//	This Function Block Performs A Linear Interpolation 
//	It Uses Multiple Data Points On Which A Line Graph Can Be Plotted
//	Between Each Two Data Points, A Line Equation Exists
//	The Linear Interpolation Formula Can Then Be Used To Find A Sensor Output Value 

FUNCTION_BLOCK Sensor_Calibration_Multipoint
VAR_INPUT
	Sensor_Input_Value		:		REAL	:=	0.0;
	
	Start_Calibration		:		BOOL	:=	FALSE;
	Reset_Calibration		:		BOOL	:=	FALSE;
END_VAR
VAR_OUTPUT
	Calibrated_Output_Value	:		REAL	:=	0.0;
END_VAR
VAR	
	// Lookup Table
	Sensor_Points			:		ARRAY[1..Calibration_Points] OF REAL	:=	[0.00, 25.00, 50.00, 75.00, 100.0];		//	Sensor Input - Will Be supplied From Analogue Scaling Block
	Reference_Points		:		ARRAY[1..Calibration_Points] OF REAL	:=	[0.00, 30.55, 58.16, 69.09, 100.0];		//	Actual Value
	
	Calibration_Index		: 		UINT;
	
	//	Linear Line Equation Variables
	X1						:		REAL	:=	0.0;
	X2						:		REAL	:=	0.0;
	Y1						:		REAL	:=	0.0;
	Y2						:		REAL	:=	0.0;	
END_VAR
VAR CONSTANT
	Calibration_Points		:		UINT	:=	5;
END_VAR

IF(Start_Calibration)THEN
	FOR Calibration_Index := 1 TO Calibration_Points DO
		//	Determine Between Which Two Data Points The Sensors Value Lies
		IF(Sensor_Input_Value >= Sensor_Points[Calibration_Index] AND Sensor_Input_Value <= Sensor_Points[Calibration_Index + 1])THEN 
			//	Determine Parameters x1, x2, y1 & y2 For Straight Line Equation
			X1	:=	Sensor_Points[Calibration_Index];
			Y1	:=	Reference_Points[Calibration_Index];
		
			X2	:=	Sensor_Points[Calibration_Index + 1];
			Y2	:=	Reference_Points[Calibration_Index + 1];
		
			Calibrated_Output_Value	:= Y1 + (Sensor_Input_Value - X1)*(Y2 - Y1)/(X2 - X1);
			EXIT;
		END_IF;
	END_FOR;
END_IF;

//	Boundary Checks
IF(Sensor_Input_Value < Sensor_Points[1])THEN
	Calibrated_Output_Value	:=	Reference_Points[1];
END_IF;

IF(Sensor_Input_Value > Sensor_Points[Calibration_Points])THEN
	Calibrated_Output_Value	:=	Reference_Points[Calibration_Points];
END_IF;

IF(Reset_Calibration)THEN
	Calibrated_Output_Value		:=	Sensor_Input_Value;
END_IF;

END_FUNCTION_BLOCK

(* stored: Version 1.1.0.1, ProductVersion 3.1.4024.15
   POU Sensor_Calibration_Multipoint: Id {a4d271ee-c364-4ccd-ad3c-bf20bb5598cc}, SpecialFunc None *)
